ABB RobotStudio station: creating_the_gripper.rsstn

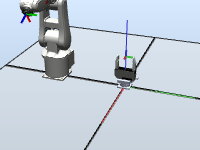
Station Station (saved by RobotStudio 6.6.7701.1025)
Layout (positions relative to the parent item):
  - IRB120_3_58__01 [mechanism, from Robots\IRB120_3_58_G_01.rslib] at (0, -541.16, 0) mm; joint values [0, 0, 0, 0, 0.5236, 0] (rad or m)
  - SmartComponent_1 [smart component, from Libraries\SCHINK_WSG_GRIPPER.rslib]
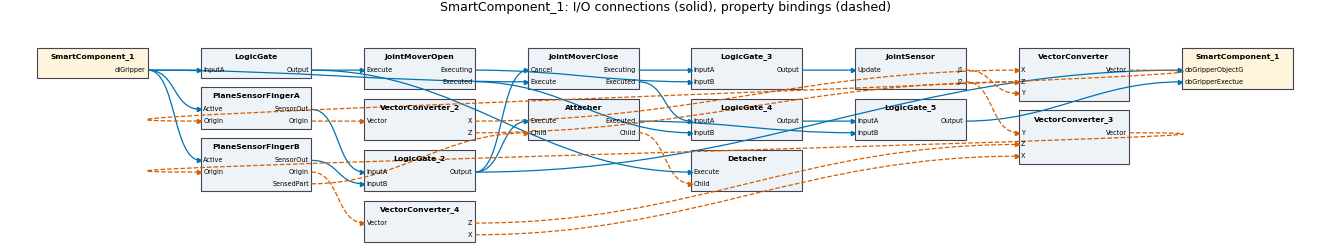
      connections:
        SmartComponent_1.diGripper -> LogicGate.InputA
        SmartComponent_1.diGripper -> PlaneSensorFingerA.Active
        SmartComponent_1.diGripper -> PlaneSensorFingerB.Active
        PlaneSensorFingerA.SensorOut -> LogicGate_2.InputA
        PlaneSensorFingerB.SensorOut -> LogicGate_2.InputB
        LogicGate_2.Output -> JointMoverClose.Cancel
        LogicGate_2.Output -> SmartComponent_1.doGripperObjectGrasped
        SmartComponent_1.diGripper -> JointMoverClose.Execute
        LogicGate.Output -> JointMoverOpen.Execute
        JointMoverClose.Executing -> LogicGate_3.InputA
        JointMoverOpen.Executing -> LogicGate_3.InputB
        LogicGate_3.Output -> JointSensor.Update
        LogicGate_2.Output -> Attacher.Execute
        LogicGate.Output -> Detacher.Execute
        JointMoverClose.Executed -> LogicGate_4.InputA
        JointMoverOpen.Executed -> LogicGate_4.InputB
        LogicGate_4.Output -> LogicGate_5.InputA
        Attacher.Executed -> LogicGate_5.InputB
        LogicGate_5.Output -> SmartComponent_1.doGripperExectued
        VectorConverter_2.X => VectorConverter.X
        VectorConverter_2.Z => VectorConverter.Z
        JointSensor.J1 => VectorConverter.Y
        PlaneSensorFingerA.Origin => VectorConverter_2.Vector
        VectorConverter.Vector => PlaneSensorFingerA.Origin
        JointSensor.J2 => VectorConverter_3.Y
        VectorConverter_4.Z => VectorConverter_3.Z
        VectorConverter_4.X => VectorConverter_3.X
        PlaneSensorFingerB.Origin => VectorConverter_4.Vector
        VectorConverter_3.Vector => PlaneSensorFingerB.Origin
        PlaneSensorFingerB.SensedPart => Attacher.Child
        Attacher.Child => Detacher.Child
    - SCHINK_WSG_GRIPPER [mechanism, from Libraries\SCHINK_WSG_GRIPPER.rslib] at (0, 0, 0) mm; joint values [0.0535, -0.0535] (rad or m)
    - PlaneSensorFingerA [smart component, from Components\PlaneSensor.rslib]
        properties: Origin=[-0.015 0.0535 0.13582]; Axis1=[0.03 0 0]; Axis2=[0 0 0.099]; SensedPart=(none)
      - _sensorPart_ [part, from Libraries\SCHINK_WSG_GRIPPER.rslib]
    - PlaneSensorFingerB [smart component, from Components\PlaneSensor.rslib]
        properties: Origin=[-0.015 -0.0535 0.13582]; Axis1=[0.03 0 0]; Axis2=[0 0 0.099]; SensedPart=(none)
      - _sensorPart_ [part, from Libraries\SCHINK_WSG_GRIPPER.rslib]
    - JointMoverClose [smart component, from Components\JointMover.rslib]
        properties: Mechanism=SCHINK_WSG_GRIPPER; Relative=false; Duration=2; J1=0; J2=0
    - JointMoverOpen [smart component, from Components\JointMover.rslib]
        properties: Mechanism=SCHINK_WSG_GRIPPER; Relative=false; Duration=2; J1=0.0535; J2=-0.0535
    - LogicGate [smart component, from Components\LogicGate.rslib]
        properties: Operator=NOT; Delay=0
    - LogicGate_2 [smart component, from Components\LogicGate.rslib]
        properties: Operator=AND; Delay=0
    - JointSensor [smart component, from Components\JointSensor.rslib]
        properties: Mechanism=SCHINK_WSG_GRIPPER; J1=0.0535; J2=-0.0535
    - LogicGate_3 [smart component, from Components\LogicGate.rslib]
        properties: Operator=OR; Delay=0
    - VectorConverter [smart component, from Components\VectorConverter.rslib]
        properties: X=-0.015; Y=0.0535; Z=0.13582; Vector=[-0.015 0.0535 0.13582]
    - VectorConverter_2 [smart component, from Components\VectorConverter.rslib]
        properties: X=-0.015; Y=0.0535; Z=0.13582; Vector=[-0.015 0.0535 0.13582]
    - VectorConverter_3 [smart component, from Components\VectorConverter.rslib]
        properties: X=-0.015; Y=-0.0535; Z=0.13582; Vector=[-0.015 -0.0535 0.13582]
    - VectorConverter_4 [smart component, from Components\VectorConverter.rslib]
        properties: X=-0.015; Y=-0.0535; Z=0.13582; Vector=[-0.015 -0.0535 0.13582]
    - Attacher [smart component, from Components\Attacher.rslib]
        properties: Parent=SCHINK_WSG_GRIPPER; Flange=0; Child=(none); Mount=false; Offset=[0 0 0]; Orientation=[0 0 0]
    - Detacher [smart component, from Components\Detacher.rslib]
        properties: Child=(none); KeepPosition=true
    - LogicGate_4 [smart component, from Components\LogicGate.rslib]
        properties: Operator=OR; Delay=0
    - LogicGate_5 [smart component, from Components\LogicGate.rslib]
        properties: Operator=OR; Delay=0
